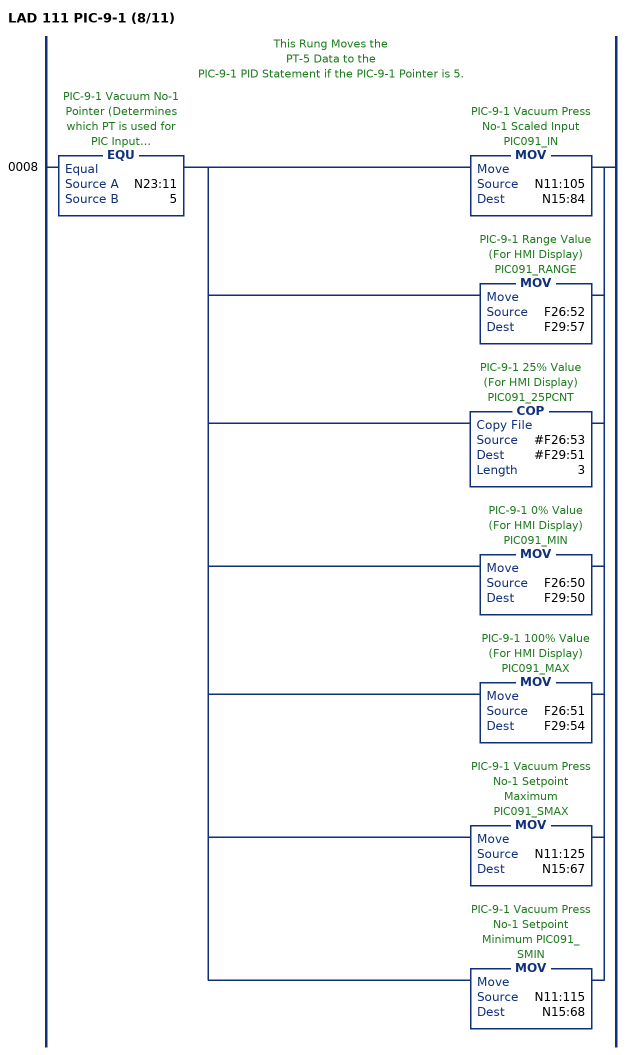
% Rung: 8 %
% This Rung Moves the
% PT-5 Data to the
% PIC-9-1 PID Statement if the PIC-9-1 Pointer is 5. %
SOR EQU N23:11 5 BST MOV N11:105 N15:84 NXB MOV F26:52 F29:57 NXB COP #F26:53 #F29:51 3 NXB MOV F26:50 F29:50 NXB MOV F26:51 F29:54 NXB MOV N11:125 N15:67 NXB MOV N11:115 N15:68 BND EOR
%   N23:11  PIC091_IN_PTR  "PIC-9-1 Vacuum No-1 Pointer (Determines which PT is used for PIC Input)" %
%   N11:105  PT05_PID_IN  "PT-05 Vacuum Transmitter No-5 PID Statement Input Value" %
%   N15:84  PIC091_IN  "PIC-9-1 Vacuum Press No-1 Scaled Input" %
%   F26:52  PT05_RANGE  "PT-5 Range Value (Max-Min)" %
%   F29:57  PIC091_RANGE  "PIC-9-1 Range Value (For HMI Display)" %
%   F26:53  PT05_25PCNT_VALUE  "PT-5 25% Range Value For HMI Display" %
%   F29:51  PIC091_25PCNT  "PIC-9-1 25% Value (For HMI Display)" %
%   F26:50  PT05_MIN  "PT-5 Minimum Value" %
%   F29:50  PIC091_MIN  "PIC-9-1 0% Value (For HMI Display)" %
%   F26:51  PT05_MAX  "PT-5 Maximum Value" %
%   F29:54  PIC091_MAX  "PIC-9-1 100% Value (For HMI Display)" %
%   N11:125  PT05_PID_MAX  "PT-05 Vacuum Transmitter No-5 PID Statement Maximum Input Value" %
%   N15:67  PIC091_SMAX  "PIC-9-1 Vacuum Press No-1 Setpoint Maximum" %
%   N11:115  PT05_PID_MIN  "PT-05 Vacuum Transmitter No-5 PID Statement Minimum Input Value" %
%   N15:68  PIC091_SMIN  "PIC-9-1 Vacuum Press No-1 Setpoint Minimum" %

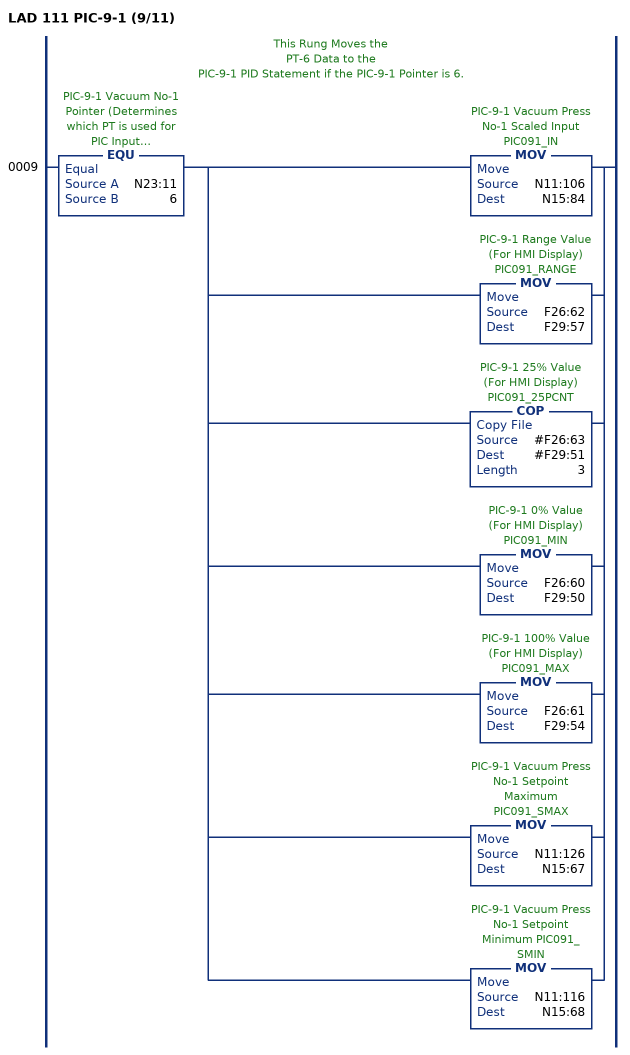
% Rung: 9 %
% This Rung Moves the
% PT-6 Data to the
% PIC-9-1 PID Statement if the PIC-9-1 Pointer is 6. %
SOR EQU N23:11 6 BST MOV N11:106 N15:84 NXB MOV F26:62 F29:57 NXB COP #F26:63 #F29:51 3 NXB MOV F26:60 F29:50 NXB MOV F26:61 F29:54 NXB MOV N11:126 N15:67 NXB MOV N11:116 N15:68 BND EOR
%   N23:11  PIC091_IN_PTR  "PIC-9-1 Vacuum No-1 Pointer (Determines which PT is used for PIC Input)" %
%   N11:106  PT06_PID_IN  "PT-06 Vacuum Transmitter No-6 PID Statement Input Value" %
%   N15:84  PIC091_IN  "PIC-9-1 Vacuum Press No-1 Scaled Input" %
%   F26:62  PT06_RANGE  "PT-6 Range Value (Max-Min)" %
%   F29:57  PIC091_RANGE  "PIC-9-1 Range Value (For HMI Display)" %
%   F26:63  PT06_25PCNT_VALUE  "PT-6 25% Range Value For HMI Display" %
%   F29:51  PIC091_25PCNT  "PIC-9-1 25% Value (For HMI Display)" %
%   F26:60  PT06_MIN  "PT-6 Minimum Value" %
%   F29:50  PIC091_MIN  "PIC-9-1 0% Value (For HMI Display)" %
%   F26:61  PT06_MAX  "PT-6 Maximum Value" %
%   F29:54  PIC091_MAX  "PIC-9-1 100% Value (For HMI Display)" %
%   N11:126  PT06_PID_MAX  "PT-06 Vacuum Transmitter No-6 PID Statement Maximum Input Value" %
%   N15:67  PIC091_SMAX  "PIC-9-1 Vacuum Press No-1 Setpoint Maximum" %
%   N11:116  PT06_PID_MIN  "PT-06 Vacuum Transmitter No-6 PID Statement Minimum Input Value" %
%   N15:68  PIC091_SMIN  "PIC-9-1 Vacuum Press No-1 Setpoint Minimum" %

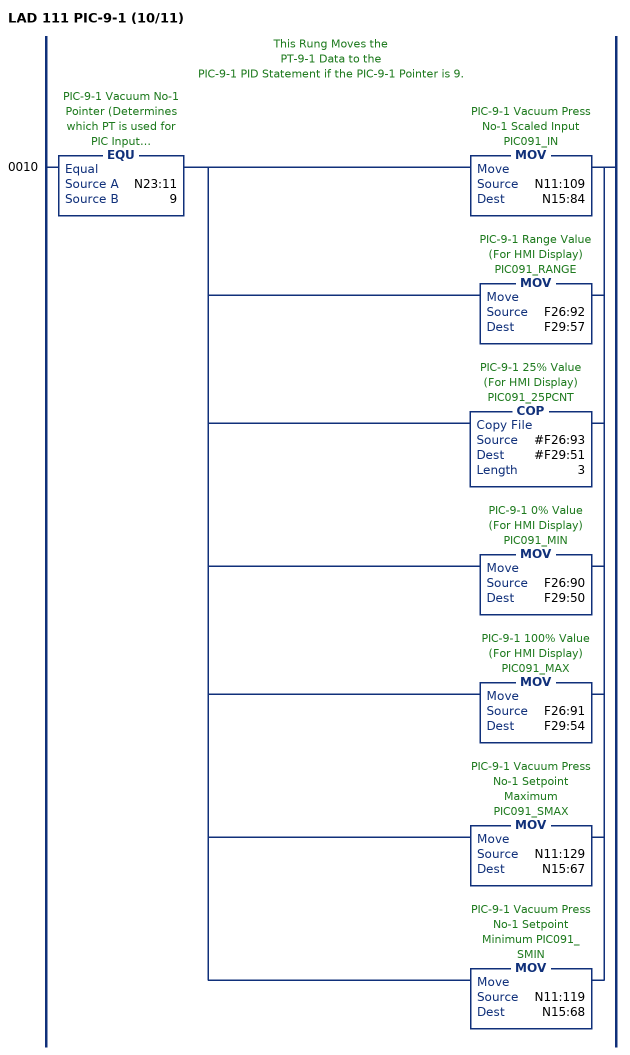
% Rung: 10 %
% This Rung Moves the
% PT-9-1 Data to the
% PIC-9-1 PID Statement if the PIC-9-1 Pointer is 9. %
SOR EQU N23:11 9 BST MOV N11:109 N15:84 NXB MOV F26:92 F29:57 NXB COP #F26:93 #F29:51 3 NXB MOV F26:90 F29:50 NXB MOV F26:91 F29:54 NXB MOV N11:129 N15:67 NXB MOV N11:119 N15:68 BND EOR
%   N23:11  PIC091_IN_PTR  "PIC-9-1 Vacuum No-1 Pointer (Determines which PT is used for PIC Input)" %
%   N11:109  PT91_PID_IN  "PT-9-1 Vacuum Transmitter PID Statement Input Value" %
%   N15:84  PIC091_IN  "PIC-9-1 Vacuum Press No-1 Scaled Input" %
%   F26:92  PT91_RANGE  "PT-9-1 Range Value (Max-Min)" %
%   F29:57  PIC091_RANGE  "PIC-9-1 Range Value (For HMI Display)" %
%   F26:93  PT91_25PCNT_VALUE  "PT-9-1 25% Range Value For HMI Display" %
%   F29:51  PIC091_25PCNT  "PIC-9-1 25% Value (For HMI Display)" %
%   F26:90  PT91_MIN  "PT-9-1 Minimum Value" %
%   F29:50  PIC091_MIN  "PIC-9-1 0% Value (For HMI Display)" %
%   F26:91  PT91_MAX  "PT-9-1 Maximum Value" %
%   F29:54  PIC091_MAX  "PIC-9-1 100% Value (For HMI Display)" %
%   N11:129  PT91_PID_MAX  "PT-9-1 Vacuum Transmitter PID Statement Maximum Input Value" %
%   N15:67  PIC091_SMAX  "PIC-9-1 Vacuum Press No-1 Setpoint Maximum" %
%   N11:119  PT91_PID_MIN  "PT-9-1 Vacuum Transmitter PID Statement Minimum Input Value" %
%   N15:68  PIC091_SMIN  "PIC-9-1 Vacuum Press No-1 Setpoint Minimum" %

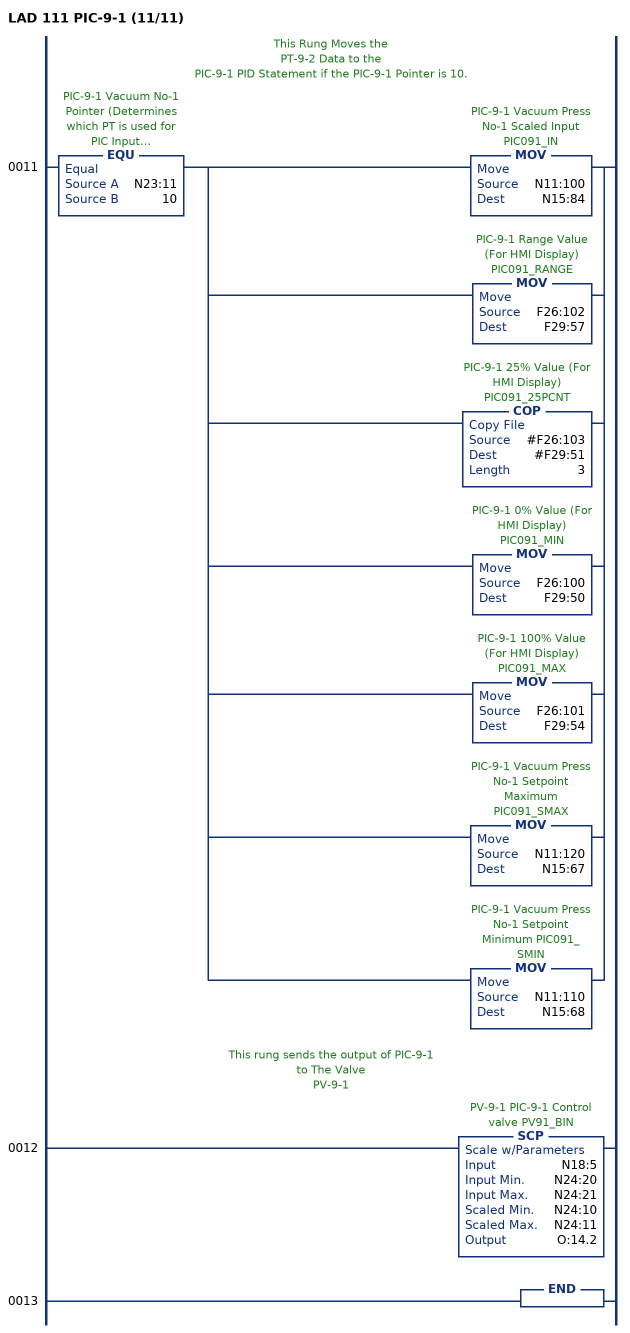
% Rung: 11 %
% This Rung Moves the
% PT-9-2 Data to the
% PIC-9-1 PID Statement if the PIC-9-1 Pointer is 10. %
SOR EQU N23:11 10 BST MOV N11:100 N15:84 NXB MOV F26:102 F29:57 NXB COP #F26:103 #F29:51 3 NXB MOV F26:100 F29:50 NXB MOV F26:101 F29:54 NXB MOV N11:120 N15:67 NXB MOV N11:110 N15:68 BND EOR
%   N23:11  PIC091_IN_PTR  "PIC-9-1 Vacuum No-1 Pointer (Determines which PT is used for PIC Input)" %
%   N11:100  PT101_PID_IN  "PT-10-1 Pressure Transmitter PID Statement Input Value" %
%   N15:84  PIC091_IN  "PIC-9-1 Vacuum Press No-1 Scaled Input" %
%   F26:102  PT101_RANGE  "PT-10-1 Range Value (Max-Min)" %
%   F29:57  PIC091_RANGE  "PIC-9-1 Range Value (For HMI Display)" %
%   F26:103  PT101_25PCNT_VALUE  "PT-10-1 25% Range Value For HMI Display" %
%   F29:51  PIC091_25PCNT  "PIC-9-1 25% Value (For HMI Display)" %
%   F26:100  PT101_MIN  "PT-10-1 Minimum Value" %
%   F29:50  PIC091_MIN  "PIC-9-1 0% Value (For HMI Display)" %
%   F26:101  PT101_MAX  "PT-10-1 Maximum Value" %
%   F29:54  PIC091_MAX  "PIC-9-1 100% Value (For HMI Display)" %
%   N11:120  PT101_PID_MAX  "PT-10-1 Pressure Transmitter PID Statement Maximum Input Value" %
%   N15:67  PIC091_SMAX  "PIC-9-1 Vacuum Press No-1 Setpoint Maximum" %
%   N11:110  PT101_PID_MIN  "PT-10-1 Pressure Transmitter PID Statement Minimum Input Value" %
%   N15:68  PIC091_SMIN  "PIC-9-1 Vacuum Press No-1 Setpoint Minimum" %
% Rung: 12 %
% This rung sends the output of PIC-9-1
% to The Valve
% PV-9-1 %
SOR SCP N18:5 N24:20 N24:21 N24:10 N24:11 O:14.2 EOR
%   N18:5  PIC091_OUT1  "PIC-9-1 Vacuum Press No-1 PID Output Value" %
%   N24:20  PID_MIN  "PID Statement Minimum Value" %
%   N24:21  PID_MAX  "PID Statement Maximum Value" %
%   N24:10  AO_MIN_NO4I  "Analog Output Minimum Value Generates 4 mA DC (To NO4I AO Module)" %
%   N24:11  AO_MAX_NO4I  "Analog Output Maximum Value Generates 20 mA DC (To NO4I AO Module)" %
%   O:14.2  PV91_BIN  "PV-9-1 PIC-9-1 Control valve" %
% Rung: 13 %
SOR END EOR

LADDER 112 "PID-10-1"    % Vacuum Control No-2 PID %
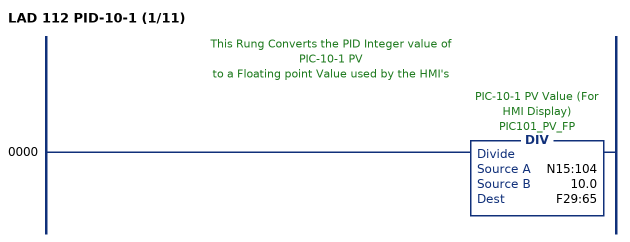
% Rung: 0 %
% This Rung Converts the PID Integer value of
% PIC-10-1 PV
% to a Floating point Value used by the HMI's %
SOR DIV N15:104 10.0 F29:65 EOR
%   N15:104  PIC101_PV  "PIC-10-1 Vacuum Press No-2 Scaled Process Variable" %
%   F29:65  PIC101_PV_FP  "PIC-10-1 PV Value (For HMI Display)" %

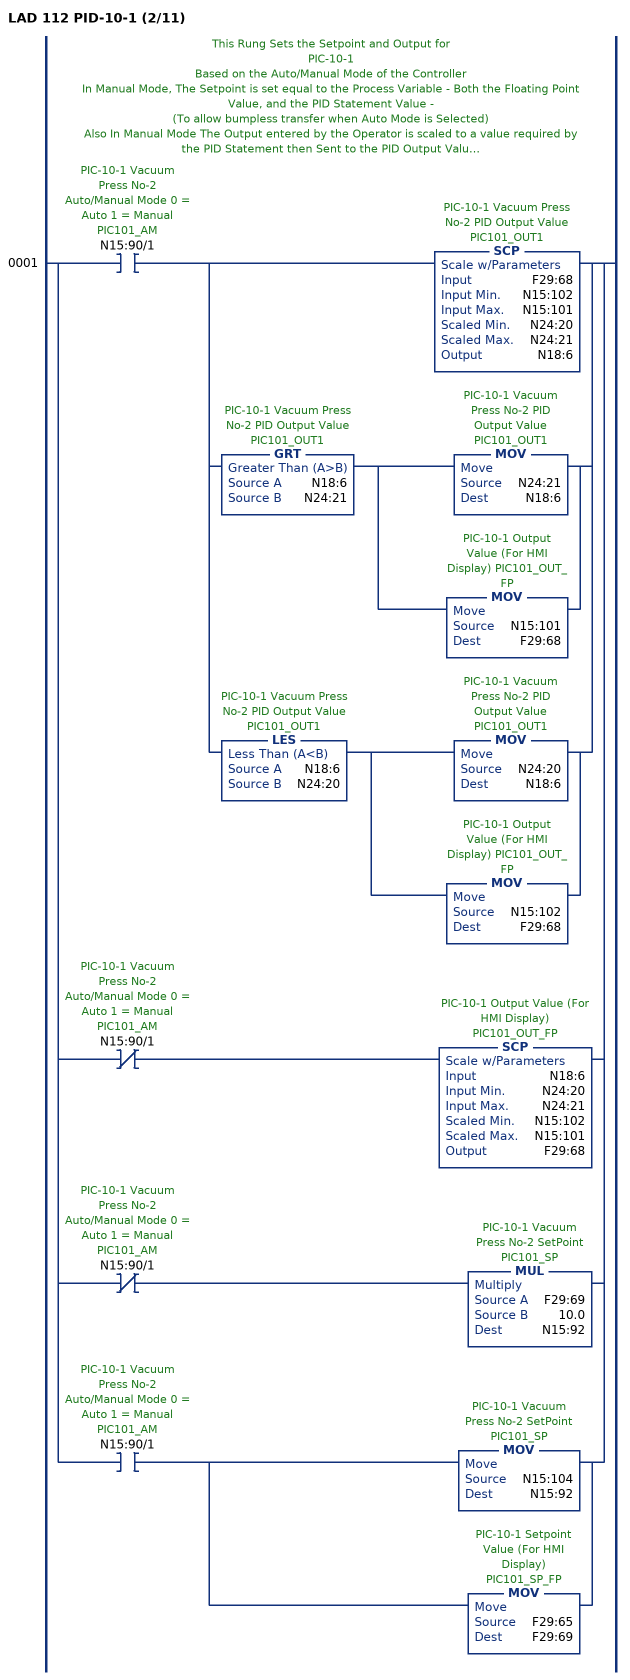
% Rung: 1 %
% This Rung Sets the Setpoint and Output for
% PIC-10-1
% Based on the Auto/Manual Mode of the Controller
% In Manual Mode, The Setpoint is set equal to the Process Variable - Both the Floating Point Value, and the PID Statement Value -
% (To allow bumpless transfer when Auto Mode is Selected)
% Also In Manual Mode The Output entered by the Operator is scaled to a value required by the PID Statement then Sent to the PID Output Value
% 
% In Auto Mode, The Setpoint is Entered by the Operator from Any HMI terminal, Multiplied by 10, and placed in the PID Statement's Setpoint Location
% Also In Auto Mode, the Output (used by the Operator) is set equal to the actual value of the pID statement
% (To allow bumpless transfer when Manual Mode is Selected) %
SOR BST XIC N15:90/1 BST SCP F29:68 N15:102 N15:101 N24:20 N24:21 N18:6 NXB GRT N18:6 N24:21 BST MOV N24:21 N18:6 NXB MOV N15:101 F29:68 BND NXB LES N18:6 N24:20 BST MOV N24:20 N18:6 NXB MOV N15:102 F29:68 BND BND NXB XIO N15:90/1 SCP N18:6 N24:20 N24:21 N15:102 N15:101 F29:68 NXB XIO N15:90/1 MUL F29:69 10.0 N15:92 NXB XIC N15:90/1 BST MOV N15:104 N15:92 NXB MOV F29:65 F29:69 BND BND EOR
%   N15:90/1  PIC101_AM  "PIC-10-1 Vacuum Press No-2 Auto/Manual Mode 0 = Auto 1 = Manual" %
%   F29:68  PIC101_OUT_FP  "PIC-10-1 Output Value (For HMI Display)" %
%   N15:102  PIC101_OMIN  "PIC-10-1 Vacuum Press No-2 Output Minimum" %
%   N15:101  PIC101_OMAX  "PIC-10-1 Vacuum Press No-2 Output Maximum" %
%   N24:20  PID_MIN  "PID Statement Minimum Value" %
%   N24:21  PID_MAX  "PID Statement Maximum Value" %
%   N18:6  PIC101_OUT1  "PIC-10-1 Vacuum Press No-2 PID Output Value" %
%   F29:69  PIC101_SP_FP  "PIC-10-1 Setpoint Value (For HMI Display)" %
%   N15:92  PIC101_SP  "PIC-10-1 Vacuum Press No-2 SetPoint" %
%   N15:104  PIC101_PV  "PIC-10-1 Vacuum Press No-2 Scaled Process Variable" %
%   F29:65  PIC101_PV_FP  "PIC-10-1 PV Value (For HMI Display)" %

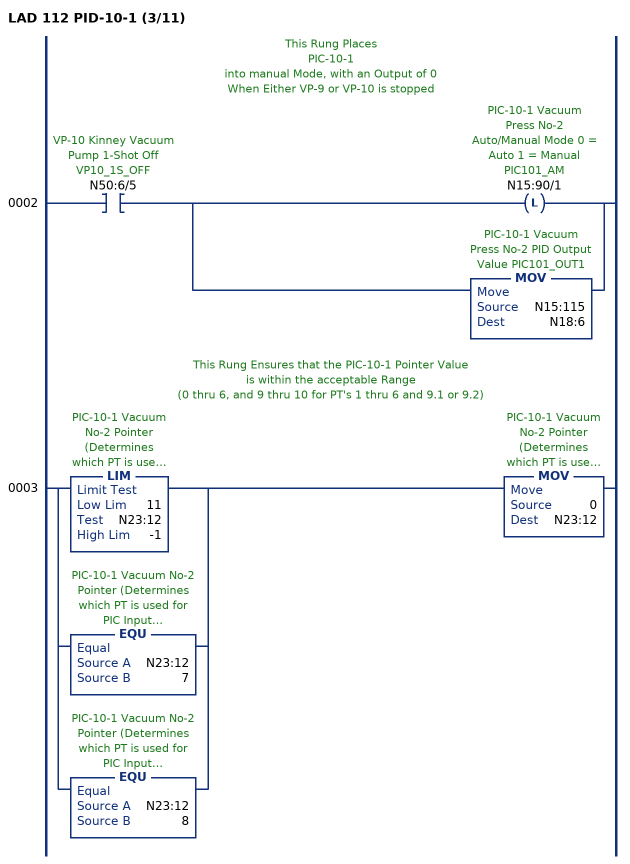
% Rung: 2 %
% This Rung Places
% PIC-10-1
% into manual Mode, with an Output of 0
% When Either VP-9 or VP-10 is stopped %
SOR XIC N50:6/5 BST OTL N15:90/1 NXB MOV N15:115 N18:6 BND EOR
%   N50:6/5  VP10_1S_OFF  "VP-10 Kinney Vacuum Pump 1-Shot Off" %
%   N15:90/1  PIC101_AM  "PIC-10-1 Vacuum Press No-2 Auto/Manual Mode 0 = Auto 1 = Manual" %
%   N15:115  PIC101_OFF_OUTPUT  "PIC-10-1 Output When VP-9 and VP-10 Are Off" %
%   N18:6  PIC101_OUT1  "PIC-10-1 Vacuum Press No-2 PID Output Value" %
% Rung: 3 %
% This Rung Ensures that the PIC-10-1 Pointer Value
% is within the acceptable Range
% (0 thru 6, and 9 thru 10 for PT's 1 thru 6 and 9.1 or 9.2) %
SOR BST LIM 11 N23:12 -1 NXB EQU N23:12 7 NXB EQU N23:12 8 BND MOV 0 N23:12 EOR
%   N23:12  PIC101_IN_PTR  "PIC-10-1 Vacuum No-2 Pointer (Determines which PT is used for PIC Input)" %

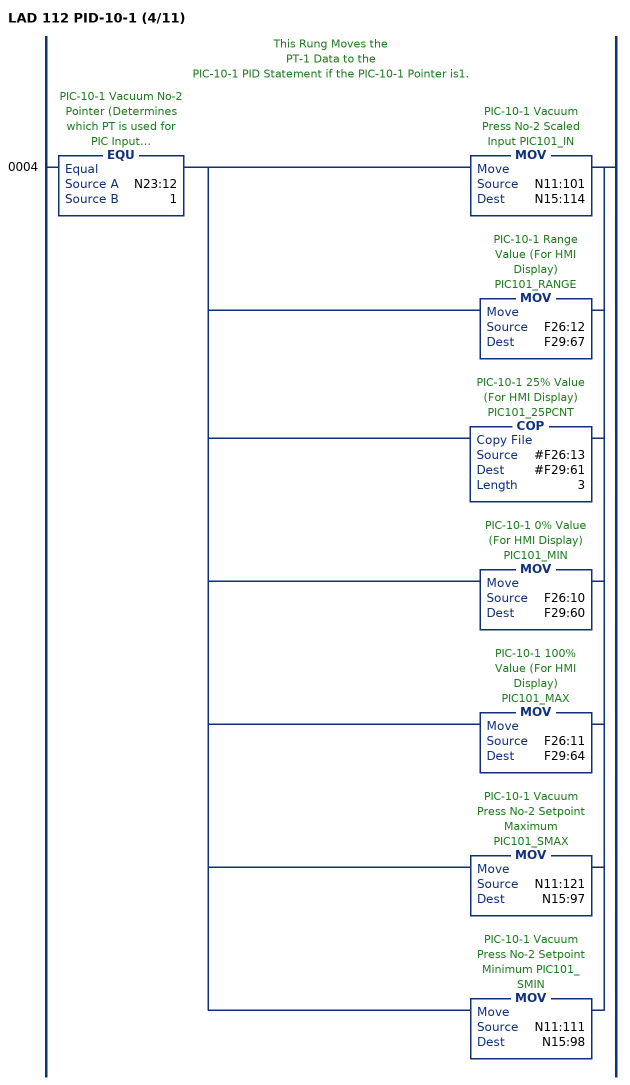
% Rung: 4 %
% This Rung Moves the
% PT-1 Data to the
% PIC-10-1 PID Statement if the PIC-10-1 Pointer is1. %
SOR EQU N23:12 1 BST MOV N11:101 N15:114 NXB MOV F26:12 F29:67 NXB COP #F26:13 #F29:61 3 NXB MOV F26:10 F29:60 NXB MOV F26:11 F29:64 NXB MOV N11:121 N15:97 NXB MOV N11:111 N15:98 BND EOR
%   N23:12  PIC101_IN_PTR  "PIC-10-1 Vacuum No-2 Pointer (Determines which PT is used for PIC Input)" %
%   N11:101  PT01_PID_IN  "PT-01 Vacuum Transmitter No-1 PID Statement Input Value" %
%   N15:114  PIC101_IN  "PIC-10-1 Vacuum Press No-2 Scaled Input" %
%   F26:12  PT01_RANGE  "PT-1 Range Value (Max-Min)" %
%   F29:67  PIC101_RANGE  "PIC-10-1 Range Value (For HMI Display)" %
%   F26:13  PT01_25PCNT_VALUE  "PT-1 25% Range Value For HMI Display" %
%   F29:61  PIC101_25PCNT  "PIC-10-1 25% Value (For HMI Display)" %
%   F26:10  PT01_MIN  "PT-1 Minimum Value" %
%   F29:60  PIC101_MIN  "PIC-10-1 0% Value (For HMI Display)" %
%   F26:11  PT01_MAX  "PT-1 Maximum Value" %
%   F29:64  PIC101_MAX  "PIC-10-1 100% Value (For HMI Display)" %
%   N11:121  PT01_PID_MAX  "PT-01 Vacuum Transmitter No-1 PID Statement Maximum Input Value" %
%   N15:97  PIC101_SMAX  "PIC-10-1 Vacuum Press No-2 Setpoint Maximum" %
%   N11:111  PT01_PID_MIN  "PT-01 Vacuum Transmitter No-1 PID Statement Minimum Input Value" %
%   N15:98  PIC101_SMIN  "PIC-10-1 Vacuum Press No-2 Setpoint Minimum" %

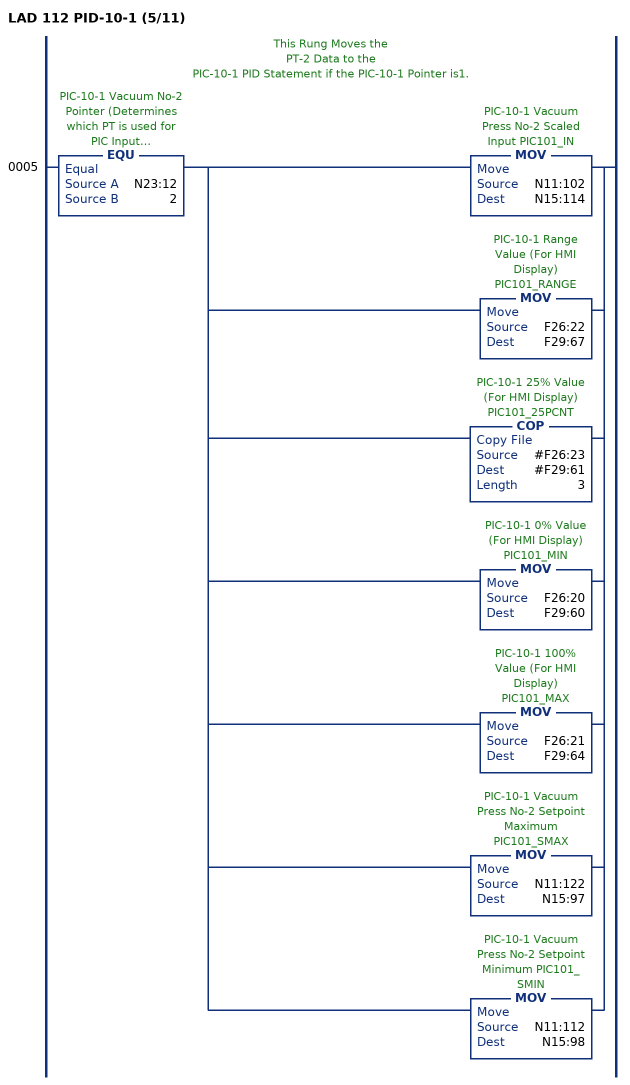
% Rung: 5 %
% This Rung Moves the
% PT-2 Data to the
% PIC-10-1 PID Statement if the PIC-10-1 Pointer is1. %
SOR EQU N23:12 2 BST MOV N11:102 N15:114 NXB MOV F26:22 F29:67 NXB COP #F26:23 #F29:61 3 NXB MOV F26:20 F29:60 NXB MOV F26:21 F29:64 NXB MOV N11:122 N15:97 NXB MOV N11:112 N15:98 BND EOR
%   N23:12  PIC101_IN_PTR  "PIC-10-1 Vacuum No-2 Pointer (Determines which PT is used for PIC Input)" %
%   N11:102  PT02_PID_IN  "PT-02 Vacuum Transmitter No-2 PID Statement Input Value" %
%   N15:114  PIC101_IN  "PIC-10-1 Vacuum Press No-2 Scaled Input" %
%   F26:22  PT02_RANGE  "PT-2 Range Value (Max-Min)" %
%   F29:67  PIC101_RANGE  "PIC-10-1 Range Value (For HMI Display)" %
%   F26:23  PT02_25PCNT_VALUE  "PT-2 25% Range Value For HMI Display" %
%   F29:61  PIC101_25PCNT  "PIC-10-1 25% Value (For HMI Display)" %
%   F26:20  PT02_MIN  "PT-2 Minimum Value" %
%   F29:60  PIC101_MIN  "PIC-10-1 0% Value (For HMI Display)" %
%   F26:21  PT02_MAX  "PT-2 Maximum Value" %
%   F29:64  PIC101_MAX  "PIC-10-1 100% Value (For HMI Display)" %
%   N11:122  PT02_PID_MAX  "PT-02 Vacuum Transmitter No-2 PID Statement Maximum Input Value" %
%   N15:97  PIC101_SMAX  "PIC-10-1 Vacuum Press No-2 Setpoint Maximum" %
%   N11:112  PT02_PID_MIN  "PT-02 Vacuum Transmitter No-2 PID Statement Minimum Input Value" %
%   N15:98  PIC101_SMIN  "PIC-10-1 Vacuum Press No-2 Setpoint Minimum" %

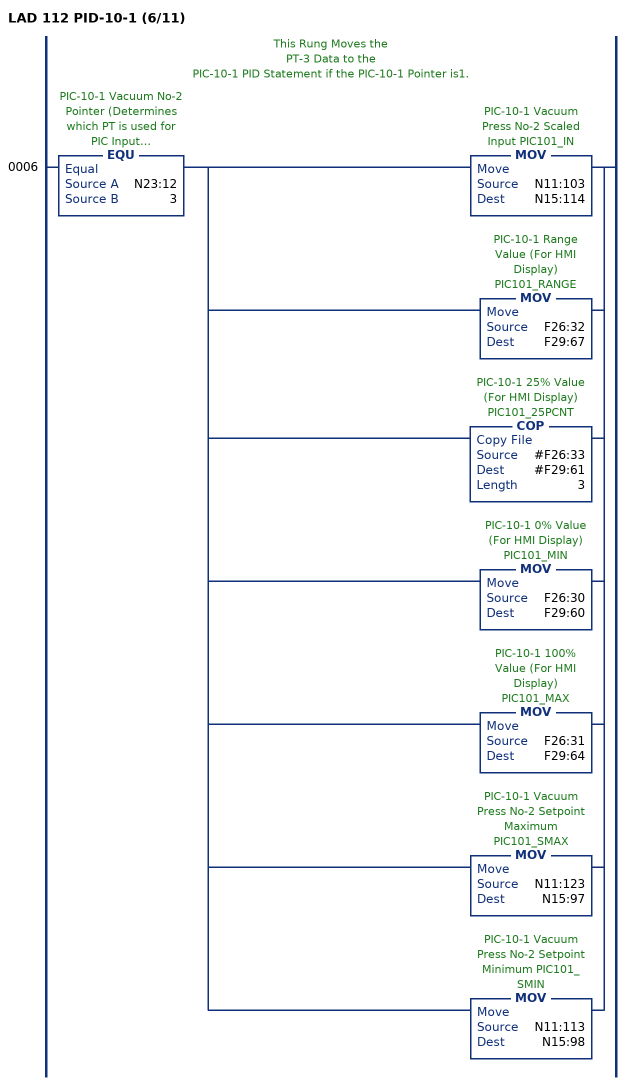
% Rung: 6 %
% This Rung Moves the
% PT-3 Data to the
% PIC-10-1 PID Statement if the PIC-10-1 Pointer is1. %
SOR EQU N23:12 3 BST MOV N11:103 N15:114 NXB MOV F26:32 F29:67 NXB COP #F26:33 #F29:61 3 NXB MOV F26:30 F29:60 NXB MOV F26:31 F29:64 NXB MOV N11:123 N15:97 NXB MOV N11:113 N15:98 BND EOR
%   N23:12  PIC101_IN_PTR  "PIC-10-1 Vacuum No-2 Pointer (Determines which PT is used for PIC Input)" %
%   N11:103  PT03_PID_IN  "PT-03 Vacuum Transmitter No-3 PID Statement Input Value" %
%   N15:114  PIC101_IN  "PIC-10-1 Vacuum Press No-2 Scaled Input" %
%   F26:32  PT03_RANGE  "PT-3 Range Value (Max-Min)" %
%   F29:67  PIC101_RANGE  "PIC-10-1 Range Value (For HMI Display)" %
%   F26:33  PT03_25PCNT_VALUE  "PT-3 25% Range Value For HMI Display" %
%   F29:61  PIC101_25PCNT  "PIC-10-1 25% Value (For HMI Display)" %
%   F26:30  PT03_MIN  "PT-3 Minimum Value" %
%   F29:60  PIC101_MIN  "PIC-10-1 0% Value (For HMI Display)" %
%   F26:31  PT03_MAX  "PT-3 Maximum Value" %
%   F29:64  PIC101_MAX  "PIC-10-1 100% Value (For HMI Display)" %
%   N11:123  PT03_PID_MAX  "PT-03 Vacuum Transmitter No-3 PID Statement Maxmium Input Value" %
%   N15:97  PIC101_SMAX  "PIC-10-1 Vacuum Press No-2 Setpoint Maximum" %
%   N11:113  PT03_PID_MIN  "PT-03 Vacuum Transmitter No-3 PID Statement Minimum Input Value" %
%   N15:98  PIC101_SMIN  "PIC-10-1 Vacuum Press No-2 Setpoint Minimum" %

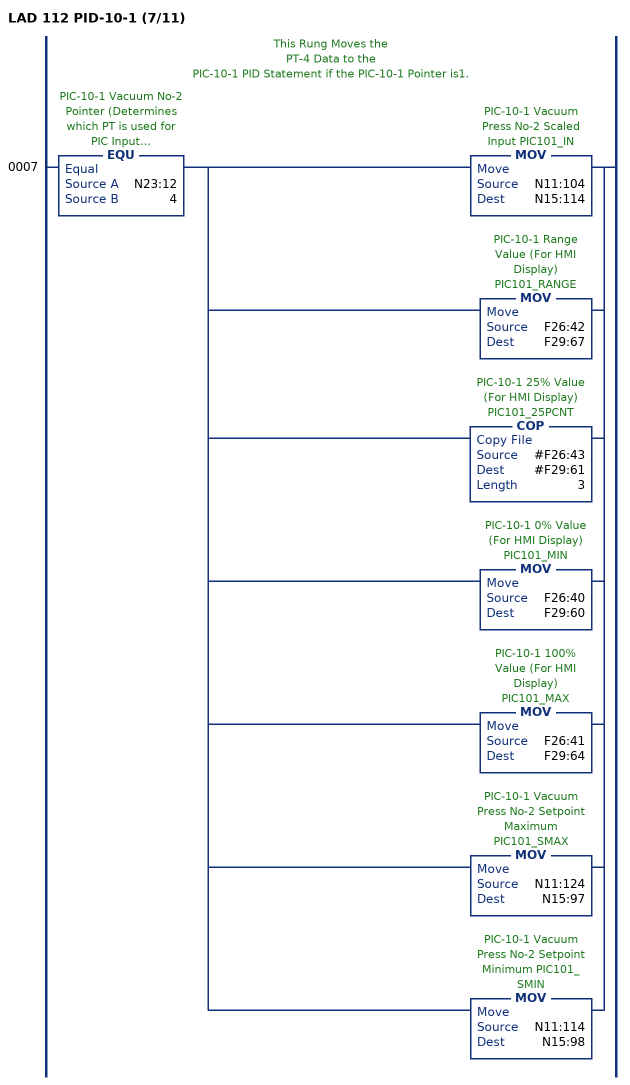
% Rung: 7 %
% This Rung Moves the
% PT-4 Data to the
% PIC-10-1 PID Statement if the PIC-10-1 Pointer is1. %
SOR EQU N23:12 4 BST MOV N11:104 N15:114 NXB MOV F26:42 F29:67 NXB COP #F26:43 #F29:61 3 NXB MOV F26:40 F29:60 NXB MOV F26:41 F29:64 NXB MOV N11:124 N15:97 NXB MOV N11:114 N15:98 BND EOR
%   N23:12  PIC101_IN_PTR  "PIC-10-1 Vacuum No-2 Pointer (Determines which PT is used for PIC Input)" %
%   N11:104  PT04_PID_IN  "PT-04 Vacuum Transmitter No-4 PID Statement Input Value" %
%   N15:114  PIC101_IN  "PIC-10-1 Vacuum Press No-2 Scaled Input" %
%   F26:42  PT04_RANGE  "PT-4 Range Value (Max-Min)" %
%   F29:67  PIC101_RANGE  "PIC-10-1 Range Value (For HMI Display)" %
%   F26:43  PT04_25PCNT_VALUE  "PT-4 25% Range Value For HMI Display" %
%   F29:61  PIC101_25PCNT  "PIC-10-1 25% Value (For HMI Display)" %
%   F26:40  PT04_MIN  "PT-4 Minimum Value" %
%   F29:60  PIC101_MIN  "PIC-10-1 0% Value (For HMI Display)" %
%   F26:41  PT04_MAX  "PT-4 Maximum Value" %
%   F29:64  PIC101_MAX  "PIC-10-1 100% Value (For HMI Display)" %
%   N11:124  PT04_PID_MAX  "PT-04 Vacuum Transmitter No-4 PID Statement Maximum Input Value" %
%   N15:97  PIC101_SMAX  "PIC-10-1 Vacuum Press No-2 Setpoint Maximum" %
%   N11:114  PT04_PID_MIN  "PT-04 Vacuum Transmitter No-4 PID Statement Minimum Input Value" %
%   N15:98  PIC101_SMIN  "PIC-10-1 Vacuum Press No-2 Setpoint Minimum" %

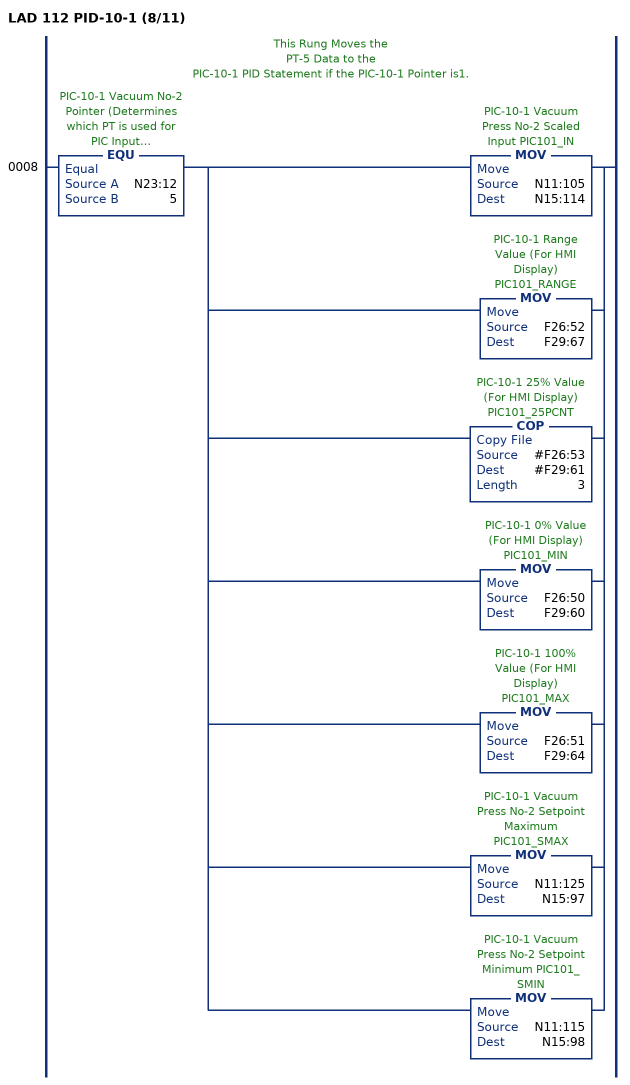
% Rung: 8 %
% This Rung Moves the
% PT-5 Data to the
% PIC-10-1 PID Statement if the PIC-10-1 Pointer is1. %
SOR EQU N23:12 5 BST MOV N11:105 N15:114 NXB MOV F26:52 F29:67 NXB COP #F26:53 #F29:61 3 NXB MOV F26:50 F29:60 NXB MOV F26:51 F29:64 NXB MOV N11:125 N15:97 NXB MOV N11:115 N15:98 BND EOR
%   N23:12  PIC101_IN_PTR  "PIC-10-1 Vacuum No-2 Pointer (Determines which PT is used for PIC Input)" %
%   N11:105  PT05_PID_IN  "PT-05 Vacuum Transmitter No-5 PID Statement Input Value" %
%   N15:114  PIC101_IN  "PIC-10-1 Vacuum Press No-2 Scaled Input" %
%   F26:52  PT05_RANGE  "PT-5 Range Value (Max-Min)" %
%   F29:67  PIC101_RANGE  "PIC-10-1 Range Value (For HMI Display)" %
%   F26:53  PT05_25PCNT_VALUE  "PT-5 25% Range Value For HMI Display" %
%   F29:61  PIC101_25PCNT  "PIC-10-1 25% Value (For HMI Display)" %
%   F26:50  PT05_MIN  "PT-5 Minimum Value" %
%   F29:60  PIC101_MIN  "PIC-10-1 0% Value (For HMI Display)" %
%   F26:51  PT05_MAX  "PT-5 Maximum Value" %
%   F29:64  PIC101_MAX  "PIC-10-1 100% Value (For HMI Display)" %
%   N11:125  PT05_PID_MAX  "PT-05 Vacuum Transmitter No-5 PID Statement Maximum Input Value" %
%   N15:97  PIC101_SMAX  "PIC-10-1 Vacuum Press No-2 Setpoint Maximum" %
%   N11:115  PT05_PID_MIN  "PT-05 Vacuum Transmitter No-5 PID Statement Minimum Input Value" %
%   N15:98  PIC101_SMIN  "PIC-10-1 Vacuum Press No-2 Setpoint Minimum" %

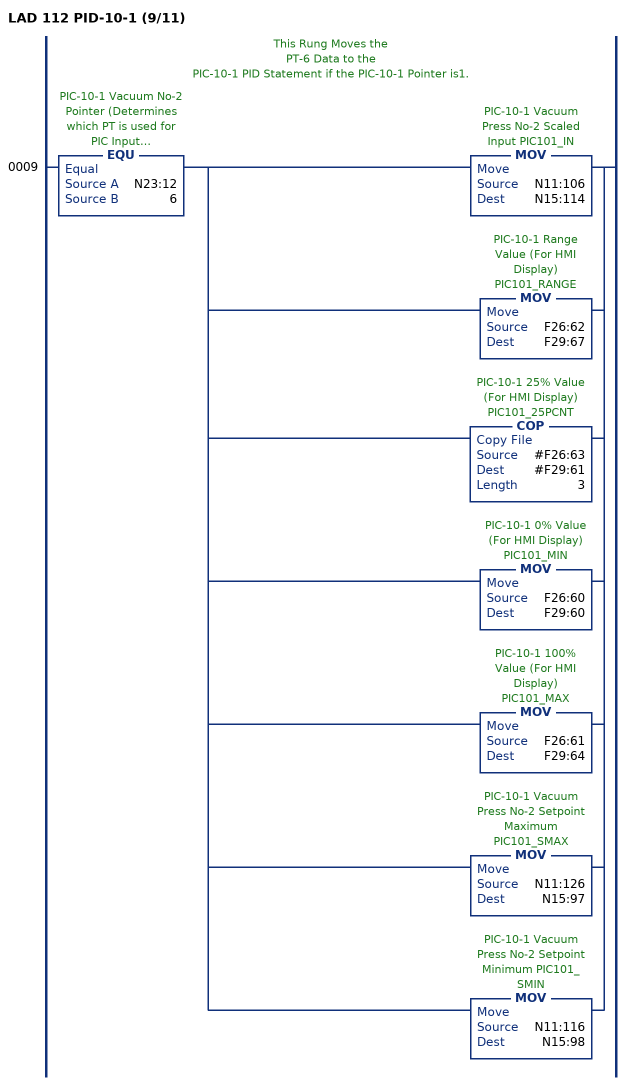
% Rung: 9 %
% This Rung Moves the
% PT-6 Data to the
% PIC-10-1 PID Statement if the PIC-10-1 Pointer is1. %
SOR EQU N23:12 6 BST MOV N11:106 N15:114 NXB MOV F26:62 F29:67 NXB COP #F26:63 #F29:61 3 NXB MOV F26:60 F29:60 NXB MOV F26:61 F29:64 NXB MOV N11:126 N15:97 NXB MOV N11:116 N15:98 BND EOR
%   N23:12  PIC101_IN_PTR  "PIC-10-1 Vacuum No-2 Pointer (Determines which PT is used for PIC Input)" %
%   N11:106  PT06_PID_IN  "PT-06 Vacuum Transmitter No-6 PID Statement Input Value" %
%   N15:114  PIC101_IN  "PIC-10-1 Vacuum Press No-2 Scaled Input" %
%   F26:62  PT06_RANGE  "PT-6 Range Value (Max-Min)" %
%   F29:67  PIC101_RANGE  "PIC-10-1 Range Value (For HMI Display)" %
%   F26:63  PT06_25PCNT_VALUE  "PT-6 25% Range Value For HMI Display" %
%   F29:61  PIC101_25PCNT  "PIC-10-1 25% Value (For HMI Display)" %
%   F26:60  PT06_MIN  "PT-6 Minimum Value" %
%   F29:60  PIC101_MIN  "PIC-10-1 0% Value (For HMI Display)" %
%   F26:61  PT06_MAX  "PT-6 Maximum Value" %
%   F29:64  PIC101_MAX  "PIC-10-1 100% Value (For HMI Display)" %
%   N11:126  PT06_PID_MAX  "PT-06 Vacuum Transmitter No-6 PID Statement Maximum Input Value" %
%   N15:97  PIC101_SMAX  "PIC-10-1 Vacuum Press No-2 Setpoint Maximum" %
%   N11:116  PT06_PID_MIN  "PT-06 Vacuum Transmitter No-6 PID Statement Minimum Input Value" %
%   N15:98  PIC101_SMIN  "PIC-10-1 Vacuum Press No-2 Setpoint Minimum" %

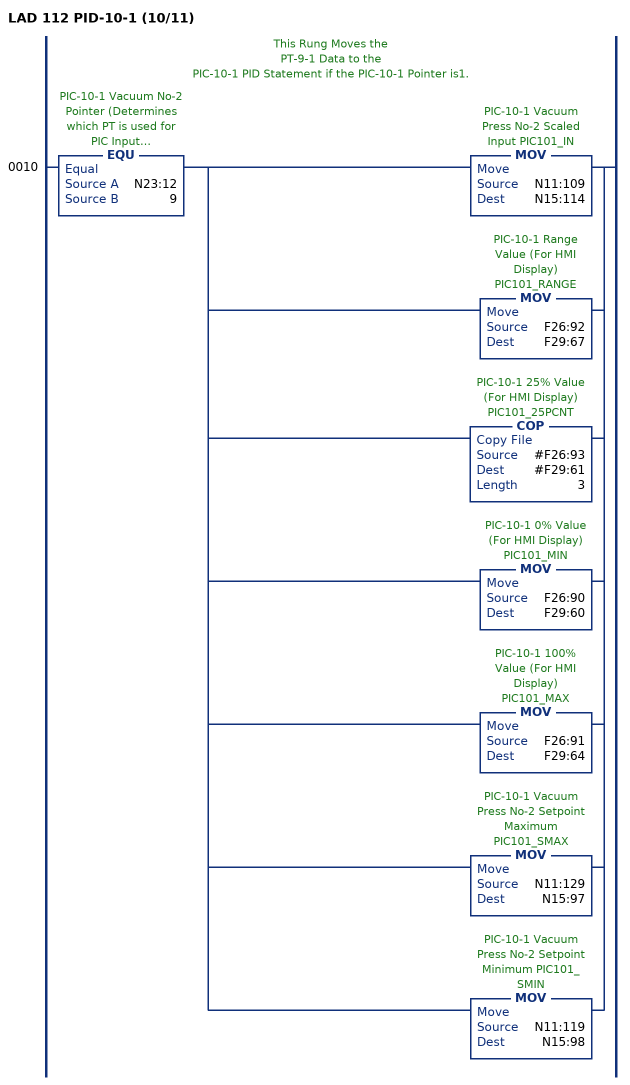
% Rung: 10 %
% This Rung Moves the
% PT-9-1 Data to the
% PIC-10-1 PID Statement if the PIC-10-1 Pointer is1. %
SOR EQU N23:12 9 BST MOV N11:109 N15:114 NXB MOV F26:92 F29:67 NXB COP #F26:93 #F29:61 3 NXB MOV F26:90 F29:60 NXB MOV F26:91 F29:64 NXB MOV N11:129 N15:97 NXB MOV N11:119 N15:98 BND EOR
%   N23:12  PIC101_IN_PTR  "PIC-10-1 Vacuum No-2 Pointer (Determines which PT is used for PIC Input)" %
%   N11:109  PT91_PID_IN  "PT-9-1 Vacuum Transmitter PID Statement Input Value" %
%   N15:114  PIC101_IN  "PIC-10-1 Vacuum Press No-2 Scaled Input" %
%   F26:92  PT91_RANGE  "PT-9-1 Range Value (Max-Min)" %
%   F29:67  PIC101_RANGE  "PIC-10-1 Range Value (For HMI Display)" %
%   F26:93  PT91_25PCNT_VALUE  "PT-9-1 25% Range Value For HMI Display" %
%   F29:61  PIC101_25PCNT  "PIC-10-1 25% Value (For HMI Display)" %
%   F26:90  PT91_MIN  "PT-9-1 Minimum Value" %
%   F29:60  PIC101_MIN  "PIC-10-1 0% Value (For HMI Display)" %
%   F26:91  PT91_MAX  "PT-9-1 Maximum Value" %
%   F29:64  PIC101_MAX  "PIC-10-1 100% Value (For HMI Display)" %
%   N11:129  PT91_PID_MAX  "PT-9-1 Vacuum Transmitter PID Statement Maximum Input Value" %
%   N15:97  PIC101_SMAX  "PIC-10-1 Vacuum Press No-2 Setpoint Maximum" %
%   N11:119  PT91_PID_MIN  "PT-9-1 Vacuum Transmitter PID Statement Minimum Input Value" %
%   N15:98  PIC101_SMIN  "PIC-10-1 Vacuum Press No-2 Setpoint Minimum" %

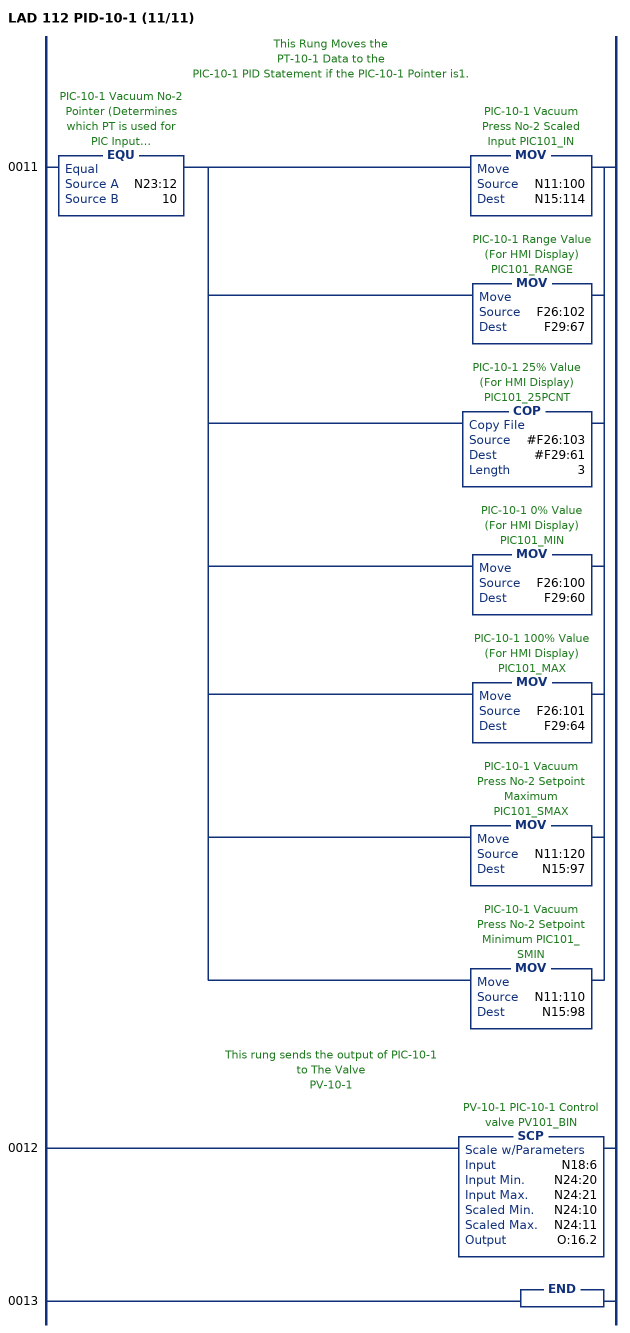
% Rung: 11 %
% This Rung Moves the
% PT-10-1 Data to the
% PIC-10-1 PID Statement if the PIC-10-1 Pointer is1. %
SOR EQU N23:12 10 BST MOV N11:100 N15:114 NXB MOV F26:102 F29:67 NXB COP #F26:103 #F29:61 3 NXB MOV F26:100 F29:60 NXB MOV F26:101 F29:64 NXB MOV N11:120 N15:97 NXB MOV N11:110 N15:98 BND EOR
%   N23:12  PIC101_IN_PTR  "PIC-10-1 Vacuum No-2 Pointer (Determines which PT is used for PIC Input)" %
%   N11:100  PT101_PID_IN  "PT-10-1 Pressure Transmitter PID Statement Input Value" %
%   N15:114  PIC101_IN  "PIC-10-1 Vacuum Press No-2 Scaled Input" %
%   F26:102  PT101_RANGE  "PT-10-1 Range Value (Max-Min)" %
%   F29:67  PIC101_RANGE  "PIC-10-1 Range Value (For HMI Display)" %
%   F26:103  PT101_25PCNT_VALUE  "PT-10-1 25% Range Value For HMI Display" %
%   F29:61  PIC101_25PCNT  "PIC-10-1 25% Value (For HMI Display)" %
%   F26:100  PT101_MIN  "PT-10-1 Minimum Value" %
%   F29:60  PIC101_MIN  "PIC-10-1 0% Value (For HMI Display)" %
%   F26:101  PT101_MAX  "PT-10-1 Maximum Value" %
%   F29:64  PIC101_MAX  "PIC-10-1 100% Value (For HMI Display)" %
%   N11:120  PT101_PID_MAX  "PT-10-1 Pressure Transmitter PID Statement Maximum Input Value" %
%   N15:97  PIC101_SMAX  "PIC-10-1 Vacuum Press No-2 Setpoint Maximum" %
%   N11:110  PT101_PID_MIN  "PT-10-1 Pressure Transmitter PID Statement Minimum Input Value" %
%   N15:98  PIC101_SMIN  "PIC-10-1 Vacuum Press No-2 Setpoint Minimum" %
% Rung: 12 %
% This rung sends the output of PIC-10-1
% to The Valve
% PV-10-1 %
SOR SCP N18:6 N24:20 N24:21 N24:10 N24:11 O:16.2 EOR
%   N18:6  PIC101_OUT1  "PIC-10-1 Vacuum Press No-2 PID Output Value" %
%   N24:20  PID_MIN  "PID Statement Minimum Value" %
%   N24:21  PID_MAX  "PID Statement Maximum Value" %
%   N24:10  AO_MIN_NO4I  "Analog Output Minimum Value Generates 4 mA DC (To NO4I AO Module)" %
%   N24:11  AO_MAX_NO4I  "Analog Output Maximum Value Generates 20 mA DC (To NO4I AO Module)" %
%   O:16.2  PV101_BIN  "PV-10-1 PIC-10-1 Control valve" %
% Rung: 13 %
SOR END EOR

LADDER 115 "PIC-28-1"    % Steam Pressure PID Controls %
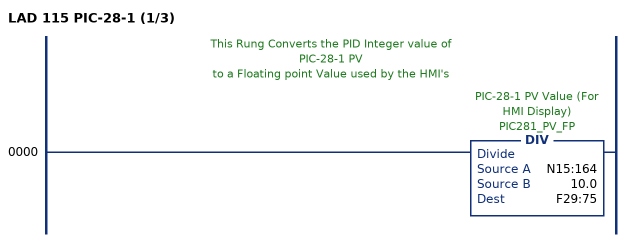
% Rung: 0 %
% This Rung Converts the PID Integer value of
% PIC-28-1 PV
% to a Floating point Value used by the HMI's %
SOR DIV N15:164 10.0 F29:75 EOR
%   N15:164  PIC281_PV  "PIC-28-1 Steam Press Scaled Process Variable" %
%   F29:75  PIC281_PV_FP  "PIC-28-1 PV Value (For HMI Display)" %

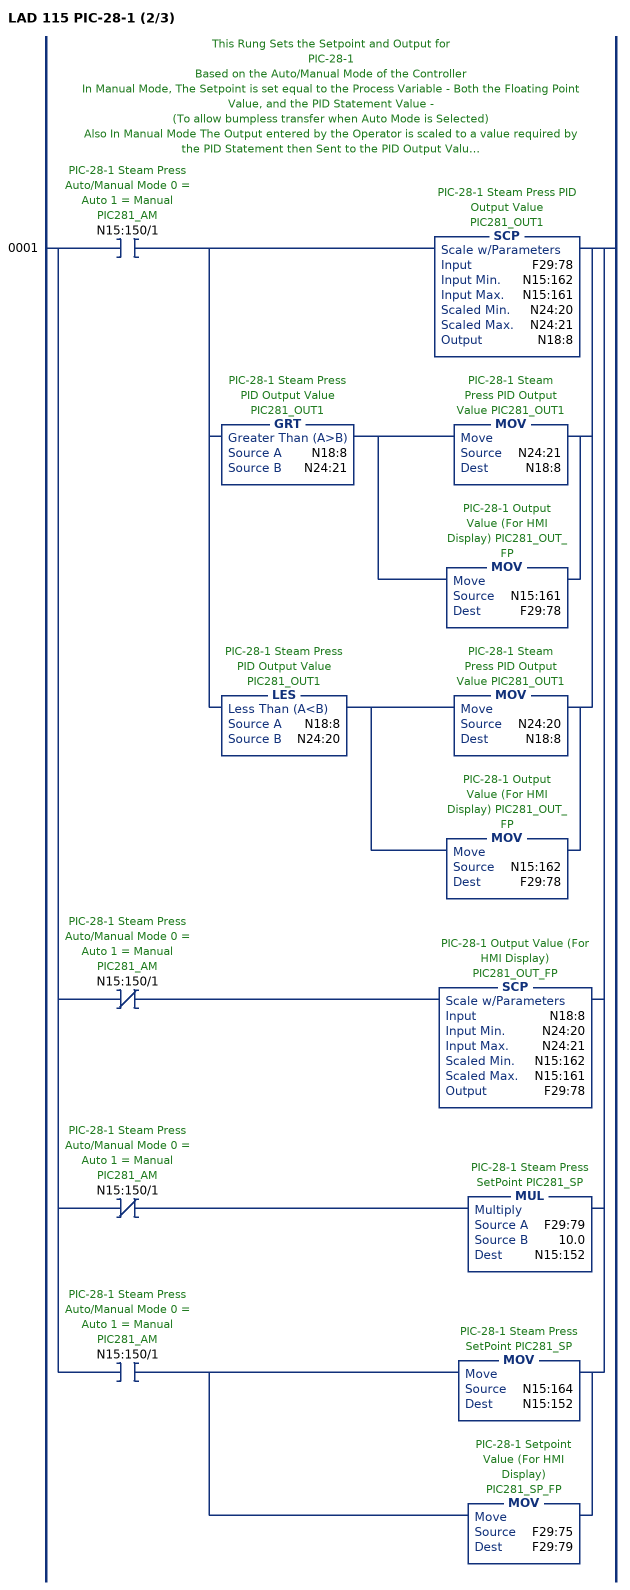
% Rung: 1 %
% This Rung Sets the Setpoint and Output for
% PIC-28-1
% Based on the Auto/Manual Mode of the Controller
% In Manual Mode, The Setpoint is set equal to the Process Variable - Both the Floating Point Value, and the PID Statement Value -
% (To allow bumpless transfer when Auto Mode is Selected)
% Also In Manual Mode The Output entered by the Operator is scaled to a value required by the PID Statement then Sent to the PID Output Value
% 
% In Auto Mode, The Setpoint is Entered by the Operator from Any HMI terminal, Multiplied by 10, and placed in the PID Statement's Setpoint Location
% Also In Auto Mode, the Output (used by the Operator) is set equal to the actual value of the pID statement
% (To allow bumpless transfer when Manual Mode is Selected) %
SOR BST XIC N15:150/1 BST SCP F29:78 N15:162 N15:161 N24:20 N24:21 N18:8 NXB GRT N18:8 N24:21 BST MOV N24:21 N18:8 NXB MOV N15:161 F29:78 BND NXB LES N18:8 N24:20 BST MOV N24:20 N18:8 NXB MOV N15:162 F29:78 BND BND NXB XIO N15:150/1 SCP N18:8 N24:20 N24:21 N15:162 N15:161 F29:78 NXB XIO N15:150/1 MUL F29:79 10.0 N15:152 NXB XIC N15:150/1 BST MOV N15:164 N15:152 NXB MOV F29:75 F29:79 BND BND EOR
%   N15:150/1  PIC281_AM  "PIC-28-1 Steam Press Auto/Manual Mode 0 = Auto 1 = Manual" %
%   F29:78  PIC281_OUT_FP  "PIC-28-1 Output Value (For HMI Display)" %
%   N15:162  PIC281_OMIN  "PIC-28-1 Steam Press Output Minimum" %
%   N15:161  PIC281_OMAX  "PIC-28-1 Steam Press Output Maximum" %
%   N24:20  PID_MIN  "PID Statement Minimum Value" %
%   N24:21  PID_MAX  "PID Statement Maximum Value" %
%   N18:8  PIC281_OUT1  "PIC-28-1 Steam Press PID Output Value" %
%   F29:79  PIC281_SP_FP  "PIC-28-1 Setpoint Value (For HMI Display)" %
%   N15:152  PIC281_SP  "PIC-28-1 Steam Press SetPoint" %
%   N15:164  PIC281_PV  "PIC-28-1 Steam Press Scaled Process Variable" %
%   F29:75  PIC281_PV_FP  "PIC-28-1 PV Value (For HMI Display)" %

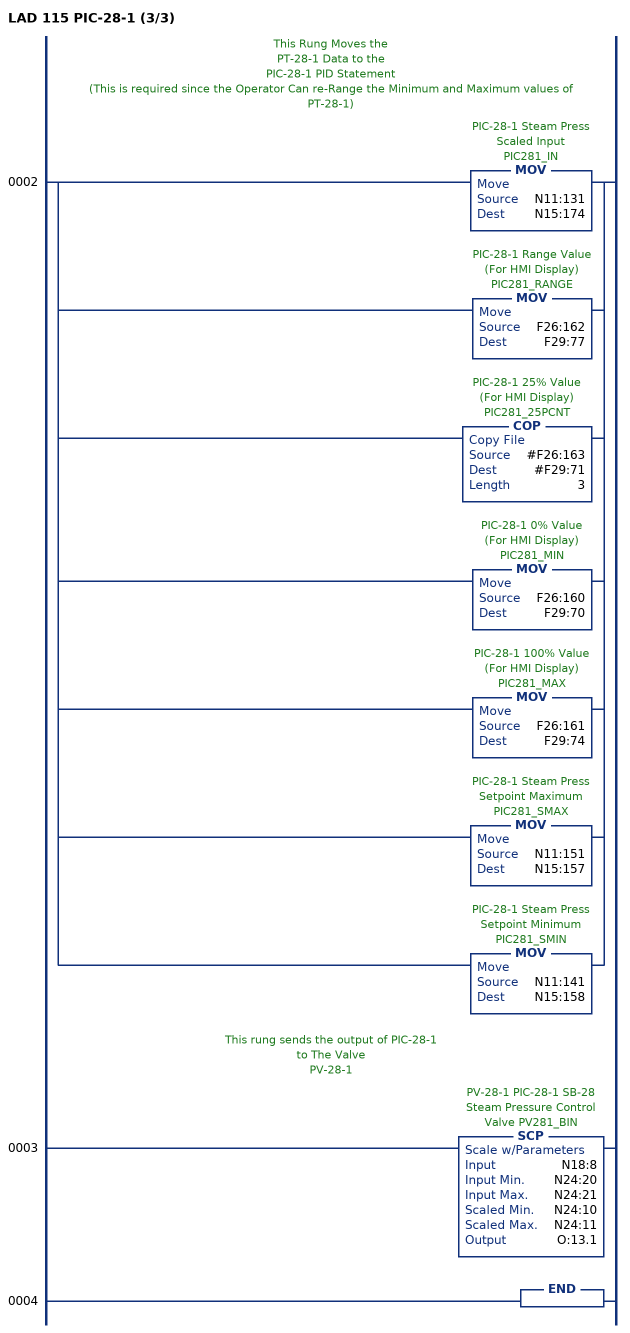
% Rung: 2 %
% This Rung Moves the
% PT-28-1 Data to the
% PIC-28-1 PID Statement
% (This is required since the Operator Can re-Range the Minimum and Maximum values of PT-28-1) %
SOR BST MOV N11:131 N15:174 NXB MOV F26:162 F29:77 NXB COP #F26:163 #F29:71 3 NXB MOV F26:160 F29:70 NXB MOV F26:161 F29:74 NXB MOV N11:151 N15:157 NXB MOV N11:141 N15:158 BND EOR
%   N11:131  PT281_PID_IN  "PT-28-1 WFE Steam Pressure PID Statement Input Value" %
%   N15:174  PIC281_IN  "PIC-28-1 Steam Press Scaled Input" %
%   F26:162  PT281_RANGE  "PT-28-1 Range Value" %
%   F29:77  PIC281_RANGE  "PIC-28-1 Range Value (For HMI Display)" %
%   F26:163  PT281_25PCNT_VALUE  "PT-28-1 25% Range Value For HMI Display" %
%   F29:71  PIC281_25PCNT  "PIC-28-1 25% Value (For HMI Display)" %
%   F26:160  PT281_MIN  "PT-28-1 Minimum Value" %
%   F29:70  PIC281_MIN  "PIC-28-1 0% Value (For HMI Display)" %
%   F26:161  PT281_MAX  "PT-28-1 Maximum Value" %
%   F29:74  PIC281_MAX  "PIC-28-1 100% Value (For HMI Display)" %
%   N11:151  PT281_PID_MAX  "PT-28-1 WFE Steam Pressure PID Statement Maximum Input Value" %
%   N15:157  PIC281_SMAX  "PIC-28-1 Steam Press Setpoint Maximum" %
%   N11:141  PT281_PID_MIN  "PT-28-1 WFE Steam Pressure PID Statement Minimum Input Value" %
%   N15:158  PIC281_SMIN  "PIC-28-1 Steam Press Setpoint Minimum" %
% Rung: 3 %
% This rung sends the output of PIC-28-1
% to The Valve
% PV-28-1 %
SOR SCP N18:8 N24:20 N24:21 N24:10 N24:11 O:13.1 EOR
%   N18:8  PIC281_OUT1  "PIC-28-1 Steam Press PID Output Value" %
%   N24:20  PID_MIN  "PID Statement Minimum Value" %
%   N24:21  PID_MAX  "PID Statement Maximum Value" %
%   N24:10  AO_MIN_NO4I  "Analog Output Minimum Value Generates 4 mA DC (To NO4I AO Module)" %
%   N24:11  AO_MAX_NO4I  "Analog Output Maximum Value Generates 20 mA DC (To NO4I AO Module)" %
%   O:13.1  PV281_BIN  "PV-28-1 PIC-28-1 SB-28 Steam Pressure Control Valve" %
% Rung: 4 %
SOR END EOR

LADDER 116 "PIC-30-1"    % Cooling Water Pressure PID Controls %
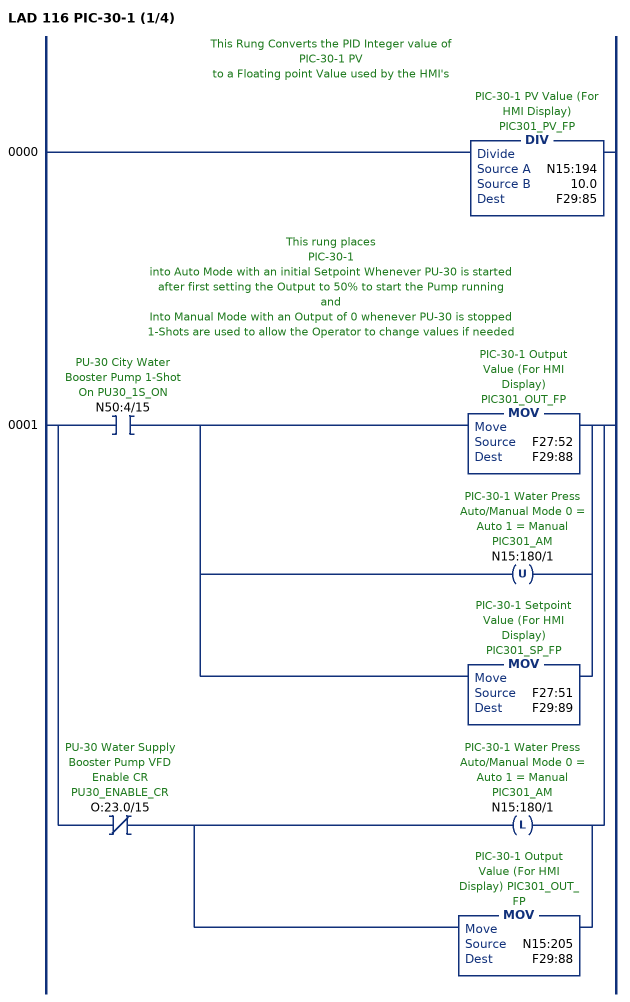
% Rung: 0 %
% This Rung Converts the PID Integer value of
% PIC-30-1 PV
% to a Floating point Value used by the HMI's %
SOR DIV N15:194 10.0 F29:85 EOR
%   N15:194  PIC301_PV  "PIC-30-1 Water Press Scaled Process Variable" %
%   F29:85  PIC301_PV_FP  "PIC-30-1 PV Value (For HMI Display)" %
% Rung: 1 %
% This rung places
% PIC-30-1
% into Auto Mode with an initial Setpoint Whenever PU-30 is started
% after first setting the Output to 50% to start the Pump running
% and
% Into Manual Mode with an Output of 0 whenever PU-30 is stopped
% 1-Shots are used to allow the Operator to change values if needed %
SOR BST XIC N50:4/15 BST MOV F27:52 F29:88 NXB OTU N15:180/1 NXB MOV F27:51 F29:89 BND NXB XIO O:23.0/15 BST OTL N15:180/1 NXB MOV N15:205 F29:88 BND BND EOR
%   N50:4/15  PU30_1S_ON  "PU-30 City Water Booster Pump 1-Shot On" %
%   F27:52  PIC301_INIT_OUTPUT  "PIC-30-1 Initial Output When Starting PU-30 Prior to placing in Auto" %
%   F29:88  PIC301_OUT_FP  "PIC-30-1 Output Value (For HMI Display)" %
%   N15:180/1  PIC301_AM  "PIC-30-1 Water Press Auto/Manual Mode 0 = Auto 1 = Manual" %
%   F27:51  PIC301_INIT_SP  "PIC-30-1 Initial Pressure Setpoint" %
%   F29:89  PIC301_SP_FP  "PIC-30-1 Setpoint Value (For HMI Display)" %
%   O:23.0/15  PU30_ENABLE_CR  "PU-30 Water Supply Booster Pump VFD Enable CR" %
%   N15:205  PIC301_OFF_OUTPUT  "PIC-30-1 Output When PU-30 Is Off" %

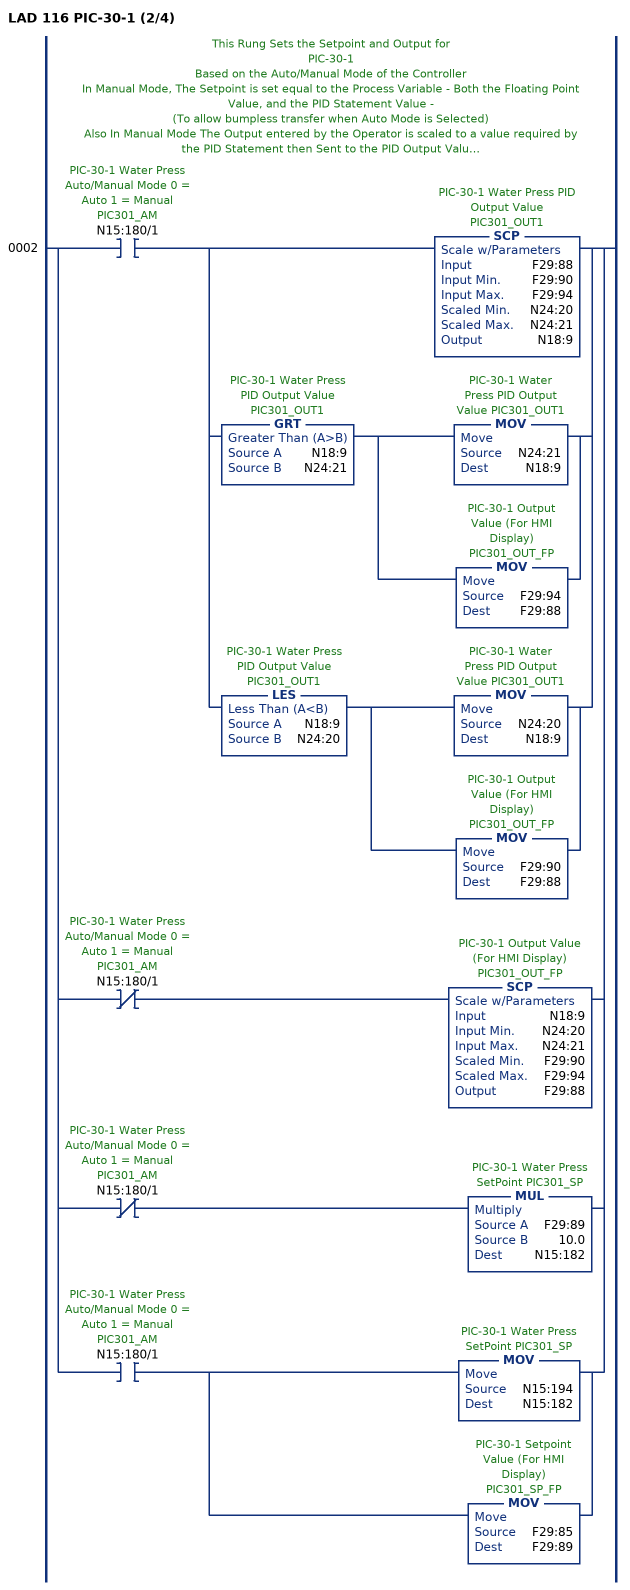
% Rung: 2 %
% This Rung Sets the Setpoint and Output for
% PIC-30-1
% Based on the Auto/Manual Mode of the Controller
% In Manual Mode, The Setpoint is set equal to the Process Variable - Both the Floating Point Value, and the PID Statement Value -
% (To allow bumpless transfer when Auto Mode is Selected)
% Also In Manual Mode The Output entered by the Operator is scaled to a value required by the PID Statement then Sent to the PID Output Value
% 
% In Auto Mode, The Setpoint is Entered by the Operator from Any HMI terminal, Multiplied by 10, and placed in the PID Statement's Setpoint Location
% Also In Auto Mode, the Output (used by the Operator) is set equal to the actual value of the pID statement
% (To allow bumpless transfer when Manual Mode is Selected) %
SOR BST XIC N15:180/1 BST SCP F29:88 F29:90 F29:94 N24:20 N24:21 N18:9 NXB GRT N18:9 N24:21 BST MOV N24:21 N18:9 NXB MOV F29:94 F29:88 BND NXB LES N18:9 N24:20 BST MOV N24:20 N18:9 NXB MOV F29:90 F29:88 BND BND NXB XIO N15:180/1 SCP N18:9 N24:20 N24:21 F29:90 F29:94 F29:88 NXB XIO N15:180/1 MUL F29:89 10.0 N15:182 NXB XIC N15:180/1 BST MOV N15:194 N15:182 NXB MOV F29:85 F29:89 BND BND EOR
%   N15:180/1  PIC301_AM  "PIC-30-1 Water Press Auto/Manual Mode 0 = Auto 1 = Manual" %
%   F29:88  PIC301_OUT_FP  "PIC-30-1 Output Value (For HMI Display)" %
%   F29:90  SIC301_MIN  "SIC-30-1 PU-30 Water Booster Pump Speed 0% Value (For HMI Display)" %
%   F29:94  SIC301_MAX  "SIC-30-1 PU-30 Water Booster Pump Speed 100% Value (For HMI Display)" %
%   N24:20  PID_MIN  "PID Statement Minimum Value" %
%   N24:21  PID_MAX  "PID Statement Maximum Value" %
%   N18:9  PIC301_OUT1  "PIC-30-1 Water Press PID Output Value" %
%   F29:89  PIC301_SP_FP  "PIC-30-1 Setpoint Value (For HMI Display)" %
%   N15:182  PIC301_SP  "PIC-30-1 Water Press SetPoint" %
%   N15:194  PIC301_PV  "PIC-30-1 Water Press Scaled Process Variable" %
%   F29:85  PIC301_PV_FP  "PIC-30-1 PV Value (For HMI Display)" %

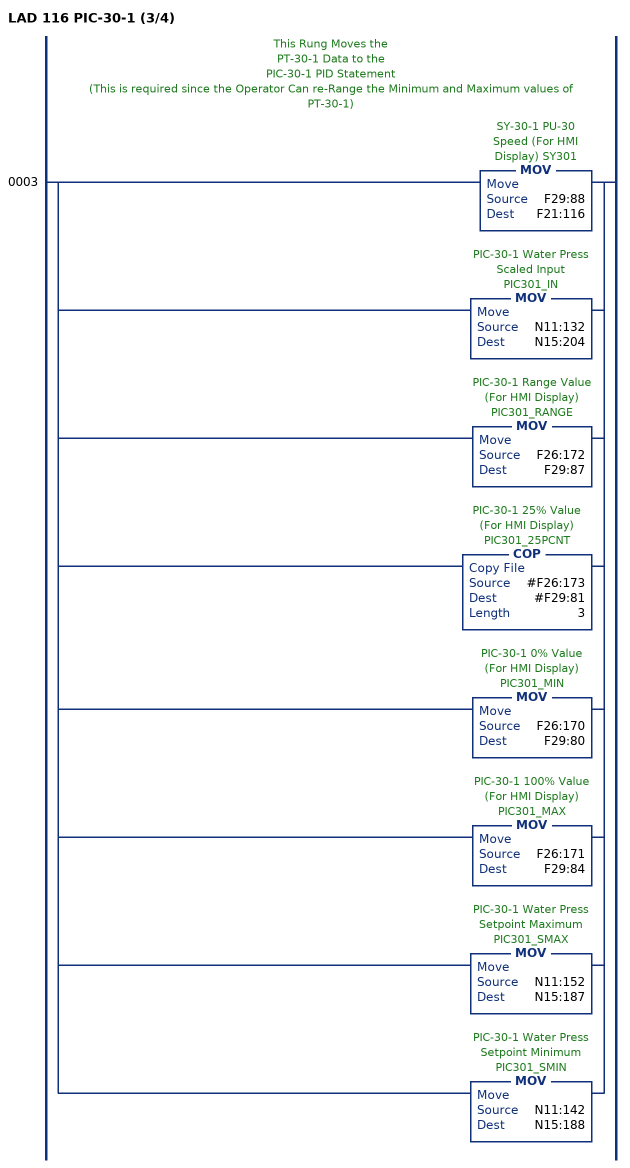
% Rung: 3 %
% This Rung Moves the
% PT-30-1 Data to the
% PIC-30-1 PID Statement
% (This is required since the Operator Can re-Range the Minimum and Maximum values of PT-30-1) %
SOR BST MOV F29:88 F21:116 NXB MOV N11:132 N15:204 NXB MOV F26:172 F29:87 NXB COP #F26:173 #F29:81 3 NXB MOV F26:170 F29:80 NXB MOV F26:171 F29:84 NXB MOV N11:152 N15:187 NXB MOV N11:142 N15:188 BND EOR
%   F29:88  PIC301_OUT_FP  "PIC-30-1 Output Value (For HMI Display)" %
%   F21:116  SY301  "SY-30-1 PU-30 Speed (For HMI Display)" %
%   N11:132  PT301_PID_IN  "PT-30-1 Cooling Water Pressure PID Statement Input Value" %
%   N15:204  PIC301_IN  "PIC-30-1 Water Press Scaled Input" %
%   F26:172  PT301_RANGE  "PT-30-1 Range Value (Max-Min)" %
%   F29:87  PIC301_RANGE  "PIC-30-1 Range Value (For HMI Display)" %
%   F26:173  PT301_25PCNT_VALUE  "PT-30-1 25% Range Value For HMI Display" %
%   F29:81  PIC301_25PCNT  "PIC-30-1 25% Value (For HMI Display)" %
%   F26:170  PT301_MIN  "PT-30-1 Minimum Value" %
%   F29:80  PIC301_MIN  "PIC-30-1 0% Value (For HMI Display)" %
%   F26:171  PT301_MAX  "PT-30-1 Maximum Value" %
%   F29:84  PIC301_MAX  "PIC-30-1 100% Value (For HMI Display)" %
%   N11:152  PT301_PID_MAX  "PT-30-1 Cooling Water Pressure PID Statement Maximum Input Value" %
%   N15:187  PIC301_SMAX  "PIC-30-1 Water Press Setpoint Maximum" %
%   N11:142  PT301_PID_MIN  "PT-30-1 Cooling Water Pressure PID Statement Minimum Input Value" %
%   N15:188  PIC301_SMIN  "PIC-30-1 Water Press Setpoint Minimum" %

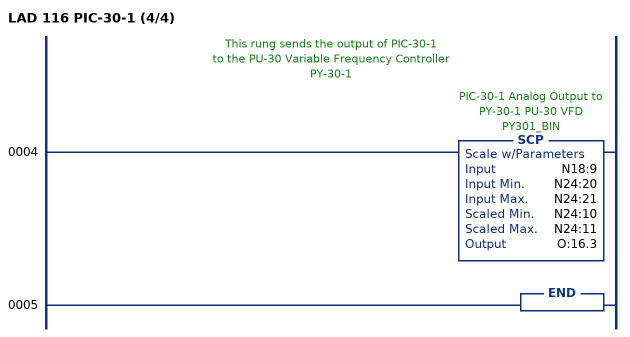
% Rung: 4 %
% This rung sends the output of PIC-30-1
% to the PU-30 Variable Frequency Controller
% PY-30-1 %
SOR SCP N18:9 N24:20 N24:21 N24:10 N24:11 O:16.3 EOR
%   N18:9  PIC301_OUT1  "PIC-30-1 Water Press PID Output Value" %
%   N24:20  PID_MIN  "PID Statement Minimum Value" %
%   N24:21  PID_MAX  "PID Statement Maximum Value" %
%   N24:10  AO_MIN_NO4I  "Analog Output Minimum Value Generates 4 mA DC (To NO4I AO Module)" %
%   N24:11  AO_MAX_NO4I  "Analog Output Maximum Value Generates 20 mA DC (To NO4I AO Module)" %
%   O:16.3  PY301_BIN  "PIC-30-1 Analog Output to PY-30-1 PU-30 VFD" %
% Rung: 5 %
SOR END EOR

LADDER 117 "PIC-46-1"    % Flash Evap Pressure Controller %
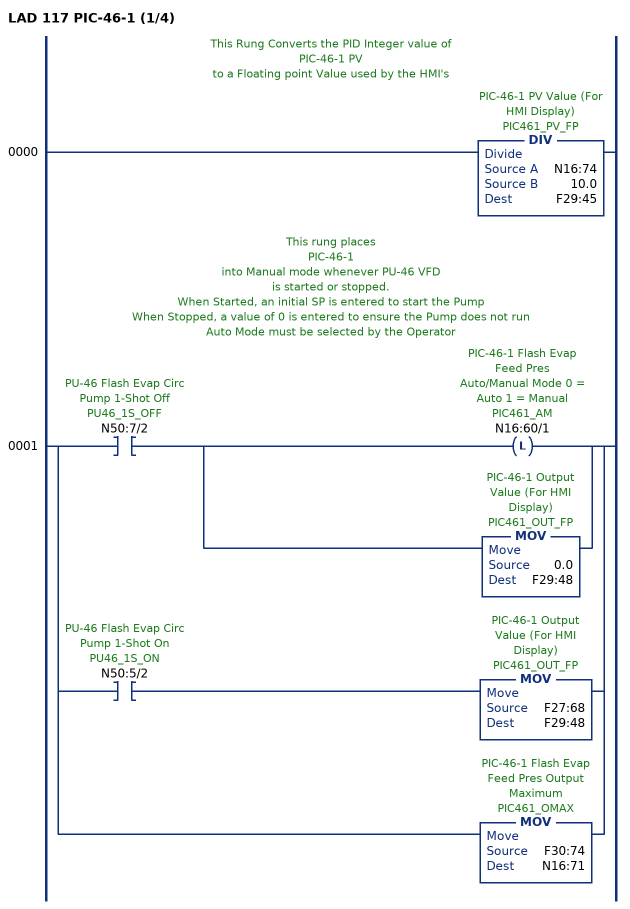
% Rung: 0 %
% This Rung Converts the PID Integer value of
% PIC-46-1 PV
% to a Floating point Value used by the HMI's %
SOR DIV N16:74 10.0 F29:45 EOR
%   N16:74  PIC461_PV  "PIC-46-1 Flash Evap Feed Pres Scaled Process Variable" %
%   F29:45  PIC461_PV_FP  "PIC-46-1 PV Value (For HMI Display)" %
% Rung: 1 %
% This rung places
% PIC-46-1
% into Manual mode whenever PU-46 VFD
% is started or stopped.
% When Started, an initial SP is entered to start the Pump
% When Stopped, a value of 0 is entered to ensure the Pump does not run
% Auto Mode must be selected by the Operator %
SOR BST XIC N50:7/2 BST OTL N16:60/1 NXB MOV 0.0 F29:48 BND NXB XIC N50:5/2 MOV F27:68 F29:48 NXB MOV F30:74 N16:71 BND EOR
%   N50:7/2  PU46_1S_OFF  "PU-46 Flash Evap Circ Pump 1-Shot Off" %
%   N16:60/1  PIC461_AM  "PIC-46-1 Flash Evap Feed Pres Auto/Manual Mode 0 = Auto 1 = Manual" %
%   F29:48  PIC461_OUT_FP  "PIC-46-1 Output Value (For HMI Display)" %
%   N50:5/2  PU46_1S_ON  "PU-46 Flash Evap Circ Pump 1-Shot On" %
%   F27:68  SIC461_INIT_SP  "SIC-46-1 Initial Speed Setpoint (Hz)" %
%   F30:74  SIC461_MAX  "SIC-46-1 PU-46 Flash Evap Circ Pump Speed at 100% Value (For HMI Display)" %
%   N16:71  PIC461_OMAX  "PIC-46-1 Flash Evap Feed Pres Output Maximum" %

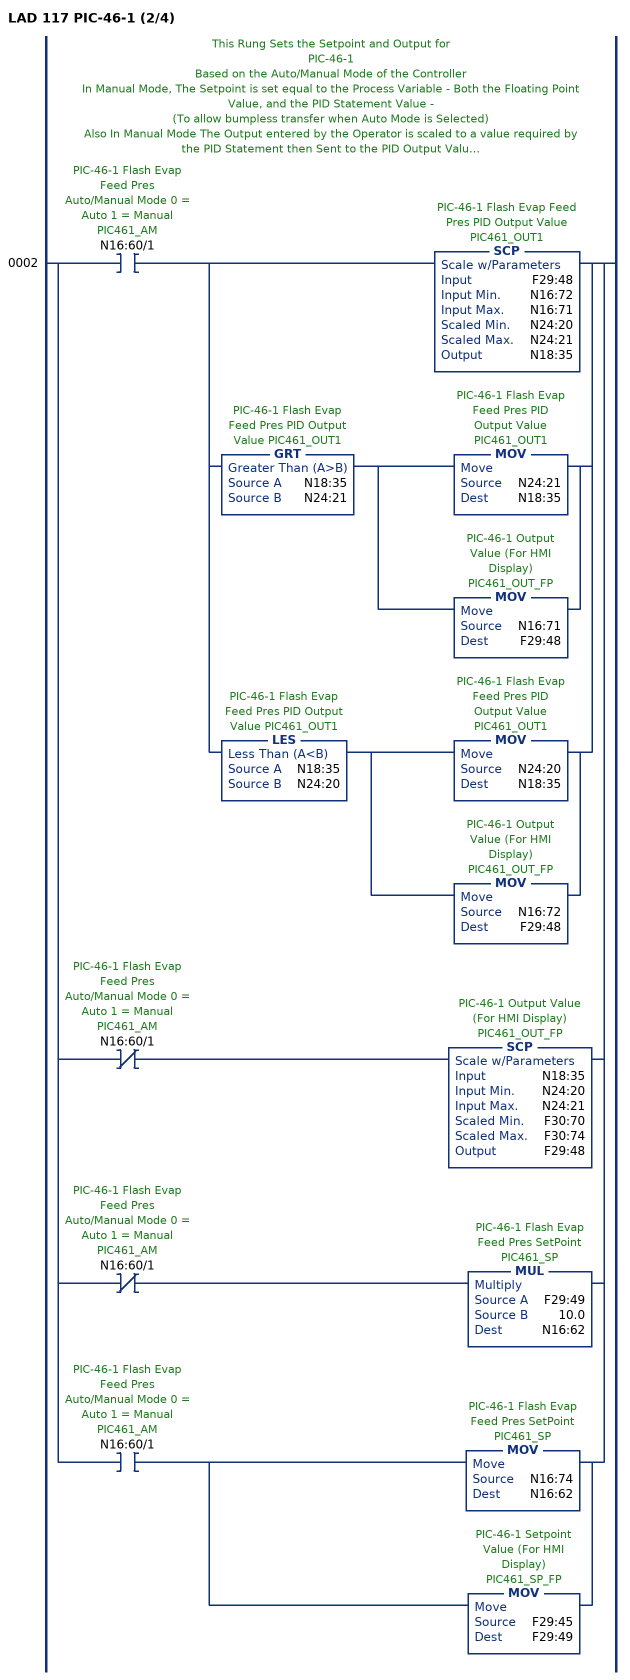
% Rung: 2 %
% This Rung Sets the Setpoint and Output for
% PIC-46-1
% Based on the Auto/Manual Mode of the Controller
% In Manual Mode, The Setpoint is set equal to the Process Variable - Both the Floating Point Value, and the PID Statement Value -
% (To allow bumpless transfer when Auto Mode is Selected)
% Also In Manual Mode The Output entered by the Operator is scaled to a value required by the PID Statement then Sent to the PID Output Value
% 
% In Auto Mode, The Setpoint is Entered by the Operator from Any HMI terminal, Multiplied by 10, and placed in the PID Statement's Setpoint Location
% Also In Auto Mode, the Output (used by the Operator) is set equal to the actual value of the pID statement
% (To allow bumpless transfer when Manual Mode is Selected) %
SOR BST XIC N16:60/1 BST SCP F29:48 N16:72 N16:71 N24:20 N24:21 N18:35 NXB GRT N18:35 N24:21 BST MOV N24:21 N18:35 NXB MOV N16:71 F29:48 BND NXB LES N18:35 N24:20 BST MOV N24:20 N18:35 NXB MOV N16:72 F29:48 BND BND NXB XIO N16:60/1 SCP N18:35 N24:20 N24:21 F30:70 F30:74 F29:48 NXB XIO N16:60/1 MUL F29:49 10.0 N16:62 NXB XIC N16:60/1 BST MOV N16:74 N16:62 NXB MOV F29:45 F29:49 BND BND EOR
%   N16:60/1  PIC461_AM  "PIC-46-1 Flash Evap Feed Pres Auto/Manual Mode 0 = Auto 1 = Manual" %
%   F29:48  PIC461_OUT_FP  "PIC-46-1 Output Value (For HMI Display)" %
%   N16:72  PIC461_OMIN  "PIC-46-1 Flash Evap Feed Pres Output Minimum" %
%   N16:71  PIC461_OMAX  "PIC-46-1 Flash Evap Feed Pres Output Maximum" %
%   N24:20  PID_MIN  "PID Statement Minimum Value" %
%   N24:21  PID_MAX  "PID Statement Maximum Value" %
%   N18:35  PIC461_OUT1  "PIC-46-1 Flash Evap Feed Pres PID Output Value" %
%   F30:70  SIC461_MIN  "SIC-46-1 PU-46 Flash Evap Circ Pump Speed 0% Value (For HMI Display)" %
%   F30:74  SIC461_MAX  "SIC-46-1 PU-46 Flash Evap Circ Pump Speed at 100% Value (For HMI Display)" %
%   F29:49  PIC461_SP_FP  "PIC-46-1 Setpoint Value (For HMI Display)" %
%   N16:62  PIC461_SP  "PIC-46-1 Flash Evap Feed Pres SetPoint" %
%   N16:74  PIC461_PV  "PIC-46-1 Flash Evap Feed Pres Scaled Process Variable" %
%   F29:45  PIC461_PV_FP  "PIC-46-1 PV Value (For HMI Display)" %

